TYPE stMachineState :
STRUCT
	Error 		: BOOL;
	CheckSafety	: BOOL;
	Aborted		: BOOL;
	Initialize	: BOOL;
	CheckToRun	: BOOL;
	Ready		: BOOL;
	Running		: BOOL;
	Stopped		: BOOL;
	ManualMode	: BOOL;
END_STRUCT
END_TYPE

(* stored: Version 1.1.0.1, ProductVersion 3.1.4024.12
   DUT stMachineState: Id {45de3a53-93c4-4338-9240-a23508b68e53} *)
